TYPE ST_HMI_DataSourceHist : 
STRUCT
	nCurrentRecordID: DINT;
	stSourceInfo: ST_HMI_DataSourceHistInfo;
	nRecordCount: DINT;
	aRecords: ARRAY [0..255] OF ST_HMI_DataSourceHistRecordInfo;
END_STRUCT
END_TYPE

(* stored: DUT ST_HMI_DataSourceHist: Id 74ee93b5-f16c-4634-9bfb-e9d64fa5e558 *)
